FUNCTION_BLOCK FB_Axis
VAR_INPUT
	// Commands
	bInJog				: BOOL;
	bInJogForward		: BOOL;
	bInJogBackward		: BOOL;
	bInPositioning		: BOOL;
	bInStop				: BOOL;
	bInReset			: BOOL;

	// Parameters
	fInVelocity			: LREAL := 1000.0;
	fInOverride			: LREAL := 100;
	fInTargetPos		: LREAL := 0;	
END_VAR
VAR_OUTPUT
	// Status
	bOutError			: BOOL;
	nOutErrorId			: UDINT;
	fOutActPosition		: DINT;
	fOutActVelocity		: DINT;
	fOutSetPosition		: LREAL;
	fOutSetVelocity		: LREAL;
	nOutAxisState		: UDINT;
	eOutAxisMode		: E_AxisMode;    
END_VAR
VAR
	// MC function blocks
	fbPower			: Tc2_MC2.MC_Power;
	fbReset			: Tc2_MC2.MC_Reset;
	fbStop			: Tc2_MC2.MC_Stop;	
	fbMoveAbs		: Tc2_MC2.MC_MoveAbsolute;
	fbJog			: Tc2_MC2.MC_Jog;
	
	// MC structures	
	stAxis			: Tc2_MC2.AXIS_REF;
	stPower			: Tc2_MC2.ST_McOutputs;
	stReset			: Tc2_MC2.ST_McOutputs;
	stStop			: Tc2_MC2.ST_McOutputs;
	stMoveAbs		: Tc2_MC2.ST_McOutputs;
	stJog			: Tc2_MC2.ST_McOutputs;
	
	// state machine
	eAxisMode		: E_AxisMode;
END_VAR

stAxis.ReadStatus();

// state machine
CASE eAxisMode OF

		E_AxisMode.INIT:
		
					fbPower.Enable := FALSE;
					fbReset.Execute := FALSE;
					fbStop.Execute := FALSE;
					fbMoveAbs.Execute := FALSE;
					fbJog.JogForward := FALSE;
					fbJog.JogBackwards := FALSE;
					eAxisMode := E_AxisMode.ENABLE;		
					
		E_AxisMode.ENABLE:					

					fbPower.Enable := TRUE;
					fbPower.Enable_Positive := TRUE;
					fbPower.Enable_Negative := TRUE;
					
					IF fbPower.Status THEN
						IF  bInStop THEN
							eAxisMode := E_AxisMode.STOP;						
						ELSIF  bInJog THEN
							eAxisMode := E_AxisMode.JOG;
						ELSIF bInPositioning THEN
							eAxisMode := E_AxisMode.POSITIONING;
						ELSIF  bInReset THEN
							eAxisMode := E_AxisMode.RESET;
						END_IF
					ELSIF fbPower.Error THEN
						eAxisMode := E_AxisMode.ERROR;						
					END_IF
					
					bOutError := fbPower.Error;
					nOutErrorId := fbPower.ErrorID;

		E_AxisMode.JOG: // Jog / manual mode with continuous speed *)					
        
					fbJog.Mode := Tc2_MC2.MC_JOGMODE_CONTINOUS;
					fbJog.Velocity := fInVelocity;
					
					IF NOT bInStop THEN
						fbJog.JogForward := bInJogForward;
						fbJog.JogBackwards := bInJogBackward;					
					END_IF
					
					IF NOT bInJog THEN
						eAxisMode := E_AxisMode.STOP;
					END_IF 
					
					(* error state *)
					IF fbJog.Error THEN
						eAxisMode := E_AxisMode.ERROR;
					END_IF
					
					bOutError := fbJog.Error;
					nOutErrorId := fbJog.ErrorID;
		
		E_AxisMode.POSITIONING: // Positioning run
				
					IF bInPositioning AND NOT fbMoveAbs.Busy THEN
						fbMoveAbs.Velocity := fInVelocity;
						fbMoveAbs.Position := fInTargetPos;
						fbMoveAbs.Execute := TRUE;
					END_IF
					
					// Wait for postioning run done
					IF fbMoveAbs.Done OR bInStop THEN
						bInPositioning := FALSE;
						fbMoveAbs.Execute := FALSE;
						eAxisMode := E_AxisMode.STOP;
					END_IF
					
					// Check if axis has an error
					IF fbMoveAbs.Error THEN
						eAxisMode := E_AxisMode.ERROR;
					END_IF
					
					bOutError := fbMoveAbs.Error;
					nOutErrorId := fbMoveAbs.ErrorID;	
					
		E_AxisMode.STOP: (* stops axis from continuos motion *)				
					fbStop.Execute := TRUE;
					IF fbStop.Active THEN
						fbStop.Execute := FALSE;
						bInStop := FALSE;
						IF fbStop.Done THEN
							bInStop := FALSE;
							eAxisMode := E_AxisMode.ENABLE;
						END_IF
					END_IF
					
					(* error state *)
					IF fbStop.Error THEN
						eAxisMode := E_AxisMode.ERROR;
					END_IF
					
					bOutError := fbStop.Error;
					nOutErrorId := fbStop.ErrorID;	

		E_AxisMode.RESET: //Reset drive to take new motion commands			

					fbReset.Execute := TRUE;
					IF fbReset.Busy THEN
						fbReset.Execute := FALSE;
						bInReset:= FALSE;
					END_IF
					IF fbReset.Done THEN
						eAxisMode := E_AxisMode.INIT;
					ELSIF fbReset.Error THEN
						eAxisMode := E_AxisMode.ERROR;
					END_IF
					
					bOutError := fbReset.Error;
					nOutErrorId := fbReset.ErrorID;

		E_AxisMode.ERROR:					

					IF stAxis.Status.Error THEN
						eAxisMode := E_AxisMode.RESET;
					ELSE
						eAxisMode := E_AxisMode.INIT;
					END_IF				

END_CASE

// Call MC function blocks
Power();
Reset();
Stop();
MoveAbs();
Jog();

// Status outputs
fOutActVelocity := TO_DINT(stAxis.NcToPlc.ActVelo);
fOutActPosition := TO_DINT(stAxis.NcToPlc.ActPos);
fOutSetVelocity := TO_LREAL(TO_DINT(stAxis.NcToPlc.SetVelo * 10000)) / 10000;
fOutSetPosition := TO_LREAL(TO_DINT(stAxis.NcToPlc.SetPos * 10000)) / 10000;
nOutAxisState := stAxis.NcToPlc.AxisState;
eOutAxisMode := eAxisMode;

ACTION Jog:
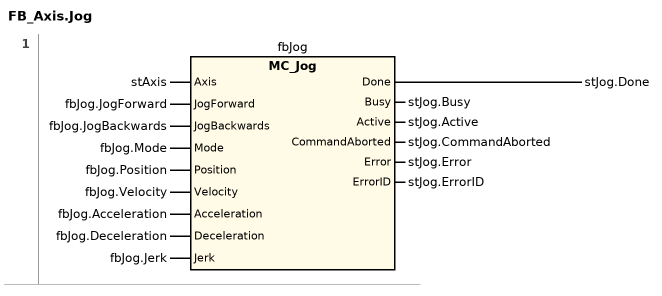
// NETWORK 1
fbJog(
    Axis := stAxis,
    JogForward := fbJog.JogForward,
    JogBackwards := fbJog.JogBackwards,
    Mode := fbJog.Mode,
    Position := fbJog.Position,
    Velocity := fbJog.Velocity,
    Acceleration := fbJog.Acceleration,
    Deceleration := fbJog.Deceleration,
    Jerk := fbJog.Jerk,
    Busy => stJog.Busy,
    Active => stJog.Active,
    CommandAborted => stJog.CommandAborted,
    Error => stJog.Error,
    ErrorID => stJog.ErrorID); // MC_Jog
stJog.Done := fbJog.Done;
END_ACTION

ACTION MoveAbs:
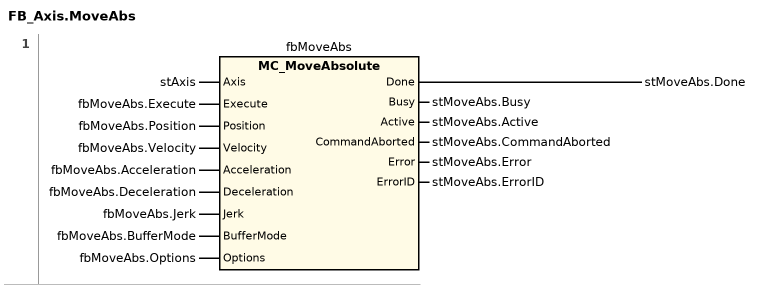
// NETWORK 1
fbMoveAbs(
    Axis := stAxis,
    Execute := fbMoveAbs.Execute,
    Position := fbMoveAbs.Position,
    Velocity := fbMoveAbs.Velocity,
    Acceleration := fbMoveAbs.Acceleration,
    Deceleration := fbMoveAbs.Deceleration,
    Jerk := fbMoveAbs.Jerk,
    BufferMode := fbMoveAbs.BufferMode,
    Options := fbMoveAbs.Options,
    Busy => stMoveAbs.Busy,
    Active => stMoveAbs.Active,
    CommandAborted => stMoveAbs.CommandAborted,
    Error => stMoveAbs.Error,
    ErrorID => stMoveAbs.ErrorID); // MC_MoveAbsolute
stMoveAbs.Done := fbMoveAbs.Done;
END_ACTION

ACTION Power:
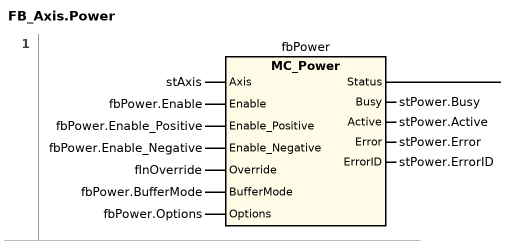
// NETWORK 1
fbPower(
    Axis := stAxis,
    Enable := fbPower.Enable,
    Enable_Positive := fbPower.Enable_Positive,
    Enable_Negative := fbPower.Enable_Negative,
    Override := fInOverride,
    BufferMode := fbPower.BufferMode,
    Options := fbPower.Options,
    Busy => stPower.Busy,
    Active => stPower.Active,
    Error => stPower.Error,
    ErrorID => stPower.ErrorID); // MC_Power
END_ACTION

ACTION Reset:
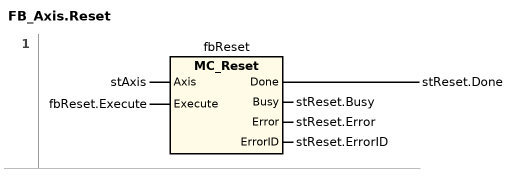
// NETWORK 1
fbReset(
    Axis := stAxis,
    Execute := fbReset.Execute,
    Busy => stReset.Busy,
    Error => stReset.Error,
    ErrorID => stReset.ErrorID); // MC_Reset
stReset.Done := fbReset.Done;
END_ACTION

ACTION Stop:
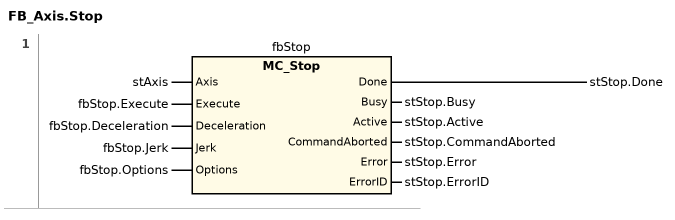
// NETWORK 1
fbStop(
    Axis := stAxis,
    Execute := fbStop.Execute,
    Deceleration := fbStop.Deceleration,
    Jerk := fbStop.Jerk,
    Options := fbStop.Options,
    Busy => stStop.Busy,
    Active => stStop.Active,
    CommandAborted => stStop.CommandAborted,
    Error => stStop.Error,
    ErrorID => stStop.ErrorID); // MC_Stop
stStop.Done := fbStop.Done;
END_ACTION

END_FUNCTION_BLOCK

(* stored: Version 1.1.0.1, ProductVersion 3.1.4022.10
   POU FB_Axis: Id {d59d1ea9-7db9-4166-9922-d0b3e52d0955}, SpecialFunc None
   Action Jog: Id {31870bcf-5036-4626-8c67-97a3615b9afe}
   Action MoveAbs: Id {d57ce96e-910b-457a-aa42-1082e62514a0}
   Action Power: Id {fb3fb0c5-4aff-48b9-80dc-20dda74bde69}
   Action Reset: Id {a22424b0-a99d-4852-860a-9c5e9d09cb9c}
   Action Stop: Id {138e6133-7c61-4f69-9086-4463a1a44903} *)
